Fanuc KAREL source: kb00073.KL

-- PROVISIONAL review KL for V770-1; original PC SHA256 586f2c03eb5e337712cc2f972b98bcab8a3c717590dbe1d37aee515cbd2393f1
-- Incomplete behavior may be omitted. Consult companion uncertainty JSON. Do not deploy.
PROGRAM KB00073
%NOLOCKGROUP
BEGIN
  -- UNRESOLVED_PC offsets 5-12; opcodes 9D,23
  -- UNRESOLVED_PC offsets 17-26; opcodes 3F,75
  -- UNRESOLVED_PC offsets 31-49; opcodes 27,22,22,2A,31
  -- UNRESOLVED_PC offsets 54-58; opcodes 7F
END KB00073
